{attribute 'Tc2GvlVarNames'}
{attribute 'strict'}
//Stato dell'ingombro dell'EndEffector
TYPE e_Stato_Ingombro_EE :
(
	EE_NOT_DEFINED				:= -1,
	EE_IN_INGOMBRO				:= 0,		(* Identifica che il Piano Di aspirazione (End-Effector) E' FUORI INGOMBRO rispetto al Punto Di prelievo *)
	EE_FUORI_INGOMBRO			:= 1		(* Identifica che il Piano Di aspirazione (End-Effector) E' IN INGOMBRO rispetto al Punto Di prelievo *)
);
END_TYPE
//  EE_NOT_DEFINED = '-1'

(* stored: Version 1.1.0.1, ProductVersion 3.1.4024.11
   EnumerationTextList e_Stato_Ingombro_EE: Id {212e671d-653b-46d9-88b2-0a3e21f92661} *)
